{attribute 'linkalways'} 
{attribute 'no_explicit_call' := 'This FB is a CLASS and must be accessed using methods or properties'}
{attribute 'enable_dynamic_creation'}
FUNCTION_BLOCK FINAL OR_SINT EXTENDS Node
VAR
	in1 : _SINT(0);
	in2 : _SINT(0);
	out : _SINT(0);
END_VAR

METHOD PUBLIC Clone : I_Node
VAR
	pNode : POINTER TO OR_SINT;
END_VAR
pNode := __NEW(OR_SINT);
Clone := pNode^;
END_METHOD

METHOD FB_init : BOOL
VAR_INPUT
	bInitRetains : BOOL; // if TRUE, the retain variables are initialized (warm start / cold start)
	bInCopyCode : BOOL;  // if TRUE, the instance afterwards gets moved into the copy code (online change)
END_VAR
AddInput('in1',THIS^.in1);
AddInput('in2',THIS^.in2);
AddOutput('out', THIS^.out);
END_METHOD

METHOD PROTECTED OnExecute
VAR
END_VAR
out.Value := in1.Value OR in2.Value;
END_METHOD

END_FUNCTION_BLOCK

(* stored: Version 1.1.0.1, ProductVersion 3.1.4024.15
   POU OR_SINT: Id {dea7fe1b-a02c-4f9a-9afe-b325a1ea3c92}, SpecialFunc None
   Folder Constructor: Id {07b6eae3-def4-4e58-80be-dad06a15427c}
   Method Clone: Id {9dc54792-378e-4b72-887f-74088ea7bc83}
   Method FB_init: Id {699c6b57-52bf-4e4a-8d06-e1669f69bb83}
   Method OnExecute: Id {de56be74-5c81-47ab-94f4-14f3bf902a82} *)
